FUNCTION_BLOCK PUBLIC TestMode
VAR_INPUT

END_VAR
VAR_OUTPUT
	TestingActive:BOOL;
END_VAR
VAR
	TestPosA: LREAL;
	TestPosB :LREAL;
	RefAxis : REFERENCE TO IDXMotor(); 
	AxisStatus : ST_AxisStatus;
	Operational :BOOL;
	InTargetPos: BOOL;
	HasJob :BOOL;
	DwellTimer: TON :=(PT:=T#5S,IN:=FALSE);
	Error :BOOL;// not used 
	TimerON: BOOL;
	Velo: LREAL;
	MoveExecute :BOOL;
	
END_VAR

//if testing active  can assume testing has begun 

//RefAxis.Status(Status =>AxisStatus); //problem
IF __ISVALIDREF(RefAxis) THEN 
	

AxisStatus := RefAxis.Status();
Operational:= AxisStatus.Operational;

IF TestingActive AND NOT Error THEN
	InTargetPos :=  AxisStatus.InTargetPosition;
	HasJob :=  AxisStatus.HasJob;
	
	IF Operational AND InTargetPos AND NOT HasJob THEN			
	 	TimerON:=TRUE;

	END_IF
	IF DwellTimer.Q THEN
		MoveExecute := TRUE;
		TimerON:=FALSE;
	END_IF

	IF ABS(RefAxis.Position()-TestPosA)<1 THEN
		RefAxis.MoveTo(Position:= TestPosB,Velocity:=Velo,Execute:=MoveExecute);
		ELSE
			RefAxis.MoveTo(Position:= TestPosA,Velocity:=Velo,Execute:=MoveExecute);
	END_IF

END_IF

IF NOT operational THEN
	TestingActive := FALSE;
END_IF

	

END_IF

DwellTimer(IN:=TimerON);

METHOD EndTest : BOOL
VAR_INPUT
	END :BOOL;
END_VAR
IF End THEN
	End:=FALSE;
	TestingActive:=FALSE;
END_IF
END_METHOD

METHOD StartTest : BOOL
VAR_INPUT
	PositionA: LREAL;
	PositionB :LREAL;
	Velocity : LREAL;
	Axis : REFERENCE TO IDXMotor();
	Dwell :TIME;
END_VAR
VAR_IN_OUT
	Execute :BOOL;
END_VAR
 IF Execute THEN
TestingActive :=TRUE;
END_IF


TestPosA := PositionA;
TestPosB := PositionB;
Velo:= Velocity;
DwellTimer.PT := dwell;
RefAxis REF= Axis;
// error if not enabled 
RefAxis.MoveTo(Position:= TestPosA,Velocity:=Velocity,Execute:=Execute);
END_METHOD

END_FUNCTION_BLOCK

(* stored: Version 1.1.0.1, ProductVersion 3.1.4024.11
   POU TestMode: Id {cc215add-2cee-463a-89db-a55b22aac16a}, SpecialFunc None
   Method EndTest: Id {3f36bde4-a7b6-49a1-aaec-56010704c723}
   Method StartTest: Id {749a70aa-672e-4cf9-8f81-4ac183f3f1bd} *)
